(* PLC project Tc2_Utilities.NT_Reboot Demo, tc3-libraries-kb TwinCAT 3.1 *)
(* stored: creationDateTime 2026-05-11T00:00:00, modificationDateTime 2026-05-11T00:00:00 *)

PROGRAM P_Demo_NT_Reboot
  VAR
    fbNT_Reboot : NT_Reboot;  (* NT_Reboot 实例 *)
    bReboot : BOOL := FALSE;
    tDelaySec : TIME := T#30S;  (* 延迟 30 秒 *)
    bBusy_ : BOOL;
    bErrFlag : BOOL;
    nErrCode : UDINT;
  END_VAR

// =============================================================================
// 场景：远程升级后自动重启。
// 价值：PLC 可触发系统重启。
// 验证：改 bReboot := TRUE 触发；30 秒后目标机器自动重启（验证前先确认非生产环境）。
// 验证步骤：
//   1. 右键 PLC 项目 → Import PLCopenXML → 选本文件
//   2. 引用 Tc2_Utilities（References → Add library）
//   3. 编译 → 登录 → 运行；按上方『验证』行的指示在线写值观察
// =============================================================================

fbNT_Reboot(
    NETID := '', START := bReboot, DELAY := UDINT_TO_DWORD(TIME_TO_UDINT(tDelaySec) / 1000),
    TMOUT := DEFAULT_ADS_TIMEOUT, BUSY => bBusy_, ERR => bErrFlag, ERRID => nErrCode
);
END_PROGRAM
